// TIA Portal V20 export
TYPE "typeMotorStarterInterface"
// stored: Access Published
   STRUCT
      et200SpMotorstarterCurrent : Array[0.."NO_OF_ET200SPMOTORSTARTER"] of Real;   // Aktuelle Werte / Current values
      et200SpMotorstarterInputs : Array[0.."NO_OF_ET200SPMOTORSTARTER"] of "LSicar_typeMotorstarterIn";   // Motorstarter Data Inputs HMI
      et200SpMotorstarterOutputs : Array[0.."NO_OF_ET200SPMOTORSTARTER"] of "LSicar_typeMotorstarterOut";   // Motorstarter Data Outputs HMI
   END_STRUCT;
END_TYPE
